FUNCTION_BLOCK EngelOutput_Test EXTENDS FB_TestSuite

SetOutputsAndVerify();

METHOD PRIVATE SetOutputsAndVerify
VAR
    out : EngelOutput;
END_VAR
TEST('SetOutputsAndVerify');

out.ManualActive(TRUE);
AssertEquals_BYTE(Expected := 2#0000_0001, Actual := out.output[39], 'SetManualActive is true');
out.ManualActive(FALSE);

out.AutomaticIsActive(TRUE);
AssertEquals_BYTE(Expected := 2#0000_0010, Actual := out.output[39], 'SetAutomaticeActive is true');
out.AutomaticIsActive(FALSE);

out.StartAutomatic(TRUE);
AssertEquals_BYTE(Expected := 2#0000_0100, Actual := out.output[39], 'SetStart is true');
out.StartAutomatic(FALSE);

out.RequestHome(TRUE);
AssertEquals_BYTE(Expected := 2#0000_1000, Actual := out.output[39], 'SetRequestHome is true');
out.RequestHome(FALSE);

out.HomeIsDone(TRUE);
AssertEquals_BYTE(Expected := 2#0001_0000, Actual := out.output[39], 'SetHomeDone is true');
out.HomeIsDone(FALSE);

out.SafetyIsClosed(TRUE);
AssertEquals_BYTE(Expected := 2#0010_0000, Actual := out.output[39], 'SetSafetyClosed is true');
out.SafetyIsClosed(FALSE);

out.RequestSafetyOpening(TRUE);
AssertEquals_BYTE(Expected := 2#0100_0000, Actual := out.output[39], 'SetSafetyOpeningRequest is true');
out.RequestSafetyOpening(FALSE);

out.SetHeartBeat(65535);
AssertEquals_BYTE(Expected := 255, Actual := out.output[1], 'Byte  1 Heartbeat shall be 255');
AssertEquals_BYTE(Expected := 255, Actual := out.output[2], 'Byte  2 Heartbeat shall be 255');

TEST_FINISHED();
END_METHOD

END_FUNCTION_BLOCK

(* stored: Version 1.1.0.1, ProductVersion 3.1.4024.12
   POU EngelOutput_Test: Id {9bb033ee-1366-4555-a805-401379e3913f}, SpecialFunc None
   Method SetOutputsAndVerify: Id {5f5a1aed-aa2f-4864-a4b7-cfd8bcdd113f} *)
